{attribute 'GeneratedUsingTerminal: EJ1957-0000-0017'}
{attribute addProperty BoxType "EJ1957-0000-0017"}
{attribute addProperty Id "Channel_1_Standard_OutputAT %Q*BOOL1Channel_2_Standard_OutputAT %Q*BOOL1Channel_3_Standard_OutputAT %Q*BOOL1Channel_4_Standard_OutputAT %Q*BOOL1"}
{attribute addProperty CRC "2128247362"}
{attribute addProperty Size "4"}
TYPE Outputs_7EDA7A42 EXTENDS OutputBase_10CEE7DE :
STRUCT
	{attribute addProperty Name "Channel_1_Standard_Output"}
	Channel_1_Standard_Output AT %Q* : BOOL;
	{attribute addProperty Name "Channel_2_Standard_Output"}
	Channel_2_Standard_Output AT %Q* : BOOL;
	{attribute addProperty Name "Channel_3_Standard_Output"}
	Channel_3_Standard_Output AT %Q* : BOOL;
	{attribute addProperty Name "Channel_4_Standard_Output"}
	Channel_4_Standard_Output AT %Q* : BOOL;
END_STRUCT
END_TYPE

(* stored: Version 1.2.0.0, ProductVersion 3.1.4024.9
   DUT Outputs_7EDA7A42: Id {e5749811-5e54-442e-9b0f-eb8bcf34a7e5} *)
